FUNCTION_BLOCK encodeIOpCdt_HMI (* Service Interface Function Block Type *)
  (* Standard: 61499-2 *)
  (* Version 0.0, 6/7/2026, Schneider Electric, template *)
  PACKAGE SE.Nereda;
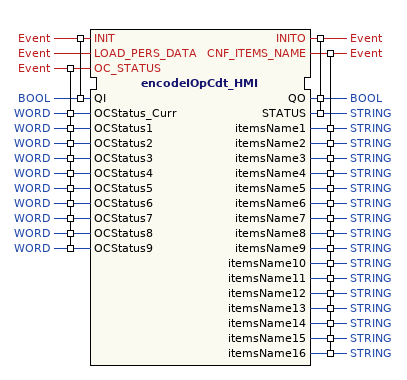
  EVENT_INPUT
    INIT WITH QI;
    LOAD_PERS_DATA;
    OC_STATUS WITH OCStatus_Curr, OCStatus1, OCStatus2, OCStatus3, OCStatus4, OCStatus5, OCStatus6, OCStatus7, OCStatus8, OCStatus9;
  END_EVENT
  EVENT_OUTPUT
    INITO WITH QO, STATUS;
    CNF_ITEMS_NAME WITH itemsName1, itemsName2, itemsName3, itemsName4, itemsName5, itemsName6, itemsName7, itemsName8, itemsName9, itemsName10, itemsName11, itemsName12, itemsName13, itemsName14, itemsName15, itemsName16;
  END_EVENT
  VAR_INPUT
    QI : BOOL;
    OCStatus_Curr : WORD;
    OCStatus1 : WORD;
    OCStatus2 : WORD;
    OCStatus3 : WORD;
    OCStatus4 : WORD;
    OCStatus5 : WORD;
    OCStatus6 : WORD;
    OCStatus7 : WORD;
    OCStatus8 : WORD;
    OCStatus9 : WORD;
  END_VAR
  VAR_OUTPUT
    QO : BOOL; (* Event Output Qualifier *)
    STATUS : STRING; (* Service Status *)
    itemsName1 : STRING;
    itemsName2 : STRING;
    itemsName3 : STRING;
    itemsName4 : STRING;
    itemsName5 : STRING;
    itemsName6 : STRING;
    itemsName7 : STRING;
    itemsName8 : STRING;
    itemsName9 : STRING;
    itemsName10 : STRING;
    itemsName11 : STRING;
    itemsName12 : STRING;
    itemsName13 : STRING;
    itemsName14 : STRING;
    itemsName15 : STRING;
    itemsName16 : STRING;
  END_VAR
  SERVICE /
    SEQUENCE 
    END_SEQUENCE
  END_SERVICE
END_FUNCTION_BLOCK
